(*~
	<docu>
	<summary>
		Provides a mechanism for inspecting status of discrete signal.	
	</summary>
	<example>										
		[!code-pas[StandardDialog](~/../TcOpen/src/TcoInspectors/src/XAE/XAE/TcoInspectorsTests/POUs/Examples/ExampleContext.TcPOU?name=StandardDialog)]		
		[!code-csharp[DialogInitialization](~/../TcOpen/src/TcoInspectors/tests/Sandbox.TcoInspectors.Wpf/MainWindowViewModel.cs?name=DialogProxyServiceInitialization)]
	</example>	
	</docu>
~*)
FUNCTION_BLOCK TcoDigitalInspector EXTENDS TcoInspector IMPLEMENTS ITcoDigitalInspector
VAR
    _data : TcoDigitalInspectorData;
END_VAR

PROPERTY CommonData : REFERENCE TO TcoInspectorData
GET
CommonData REF= _data;
END_GET
END_PROPERTY

(*~
<docu>
<summary>
	Gets data of this inspector.
</summary>
</docu>
~*)
PROPERTY Data : REFERENCE TO TcoDigitalInspectorData
GET
Data REF= _data;
END_GET
END_PROPERTY

(*~
<docu>
<summary>
	Inspects the signal and evaluates that it matches the value set in `RequiredStatus`.
</summary>
<returns>
	Returns the interface with information about the state of inspection.
</returns>
</docu>
~*)
METHOD Inspect : IInspector
VAR_INPUT
    Status : BOOL;
END_VAR
Inspect := THIS^;

_inspectorTask.InspectionData REF= _data;

OnEnterInspection();

IF(IsOverinspected())THEN
	RETURN;
END_IF


_inspectorTask.Invoke();

IF (_inspectorTask.Execute()) THEN
    IF (_data.IsByPassed) THEN
        _data.Result    := eInspectorResult.Bypassed;
        _data.TimeStamp := Context.RealTimeClock.NowLocal();
        _inspectorTask.DoneWhen(TRUE);
        RETURN;
    END_IF

    _data.Result := eInspectorResult.Running;
    _inspectorTask._failTimer(IN := TRUE, PT := _data.FailTime);
    _inspectorTask._passTimer(IN := Status = _data.RequiredStatus, PT := _data.PassTime);
    _data.DetectedStatus := Status;    
  
    IF(_inspectorTask._failTimer.Q OR _inspectorTask._passTimer.Q) THEN	  
     		_inspectorTask.DoneWhen(TRUE);
			OnDone();
	END_IF;	
END_IF;
END_METHOD

(*~
	<docu>
		<summary>
			Executes when task reaches the ```Done``` state .
		</summary>			
	</docu>	
~*)
METHOD PROTECTED OnDone
IF (_data.Result = eInspectorResult.Failed) THEN
     _data.DetectedStatus := NOT _data.RequiredStatus;
END_IF
END_METHOD

METHOD WithCoordinator : ITcoDigitalInspector
VAR_INPUT
	inCoordinator : TcoCore.ITcoCoordinator;
END_VAR
_WithCoordinator(inCoordinator);
WithCoordinator := THIS^;
END_METHOD

END_FUNCTION_BLOCK

(* stored: Version 1.1.0.1, ProductVersion 3.1.4024.9
   POU TcoDigitalInspector: Id {b1413ab6-cf32-03b8-31af-46a8ec8720ab}, SpecialFunc None
   Property CommonData: Id {b45e0a39-37d2-0d84-323d-7324b429b3a2}
   Get Get: Id {2673f909-9f9c-0376-1ac6-0f51ac4a44b2}
   Property Data: Id {b0f00037-c485-0f58-3a2e-35a438d55d1b}
   Get Get: Id {9d81d3dd-148f-0c90-116b-61d78b860286}
   Method Inspect: Id {304a74e1-ec39-09fd-0ecf-8a74644a243b}
   Method OnDone: Id {a41dc408-1e34-0f67-0765-b3b3943d0f0d}
   Method WithCoordinator: Id {943d74b5-be94-00d9-004e-ca370a1acdd8} *)
